Staubli VAL3: _tcycle.pgx

public program _tcycle()
begin
  while true

  endWhile
end
